// TIA Portal V20 export
TYPE "typeEMIdentRf"
// stored: Access Published
   STRUCT
      identRfEM : Array[0.."NO_OF_EM"] of "typeIdentRfHmi";
   END_STRUCT;
END_TYPE
